# B&R Automation Studio project datmod
Automation Studio 4.3.6.57 SP; Default project

## Configuration Simulation

CPU , AutomationRuntime G4.34, Build 4.1.2, Vc V4.34.2

### Task classes (Cpu.sw)
```
Cyclic#1 (cycle 100000 us, tolerance 10000000 us):
  recipe <- recipe.prg
Binaries: ashwd, sysconf, asfw, arconfig, iomap
Libraries: AsIecCon, astime, datmodHand, DataObj, runtime
```

### Hardware
```
PLC1 : PC_any v1.1.0.0 (OrderNumber=PC)
  VolatileGlobalPvSize = 4096
  XLinkUseDefault = 0
  Cyclic1Duration = 100000
  Cyclic1Tolerance = 10000000
  Cyclic2Duration = 200000
  Cyclic2Tolerance = 10000000
  Cyclic3Duration = 500000
  Cyclic3Tolerance = 10000000
  Cyclic4Duration = 1000000
  Cyclic4Tolerance = 10000000
  Cyclic5Duration = 2000000
  Cyclic5Tolerance = 10000000
  Cyclic6Duration = 3000000
  Cyclic6Tolerance = 12000000
  Cyclic7Duration = 4000000
  Cyclic7Tolerance = 12000000
  Cyclic8Duration = 5000000
  Cyclic8Tolerance = 30000000
```

## Logical view

Binary libraries used (declarations not repeated): DataObj, Runtime, Operator, AsIecCon, astime

### Program Logical/recipe (IEC) - sample program

#### recipe.st - Implementation code
```iecst
PROGRAM _INIT

recipe1.milk := 0.4;
recipe1.name := 'espresso';
recipe1.sugar := 1;

//
END_PROGRAM

PROGRAM _CYCLIC

	CASE step OF
		0: (* store data *)
		recipeHandling.para.pData := ADR(recipe1);
		recipeHandling.para.dataLen := SIZEOF(recipe1);
		recipeHandling.para.memType := doUSRROM;
		recipeHandling.para.name := 'recipe00';
		recipeHandling.para.overwriteExisting := 1;
		recipeHandling.cmd.save := 1;
		step := 1;

		1: (* load data *)
		IF recipeHandling.status.ok THEN
			recipeHandling.para.pData := ADR(recipe2);
			recipeHandling.para.dataLen := SIZEOF(recipe1);
			recipeHandling.para.memType := doUSRROM;
			recipeHandling.para.name := 'recipe00';
			recipeHandling.cmd.load := 1;
			step := 2;
		END_IF

		2:

	END_CASE

	(* call function *)
	datmodHand( recipeHandling );

END_PROGRAM
```

#### recipe.typ - Local data types
```iecst
TYPE
	myRecipe : 	STRUCT
		sugar : USINT;
		milk : REAL;
		name : STRING[20];
	END_STRUCT;
END_TYPE
```

#### recipe.var - Local variables
```iecst
VAR
	step : USINT := 0;
	recipe2 : myRecipe := (0);
	recipe1 : myRecipe := (0);
	recipeHandling : datmodHand_typ := (0);
END_VAR
```

### Package Logical/Libraries - Global libraries

### Library Logical/Libraries/datmodHand (IEC) - simple data module handling

#### datmodHand.typ - Exported data types
```iecst
TYPE
	datmodHandPara_typ : 	STRUCT
		name : STRING[10]; (*name of data module*)
		overwriteExisting : BOOL; (*overwrite existing module*)
		pData : UDINT; (*pointer to data buffer*)
		dataLen : UDINT; (*length of data*)
		memType : USINT; (*target memory in which the data object is to be saved,  e.g. doTEMP, doUSRRAM, doUSRROM, ...*)
	END_STRUCT;
	datmodHandCmd_typ : 	STRUCT  (*1 = execute, 2 = busy*)
		load : BOOL; (*load module*)
		save : BOOL; (*save data to module*)
		delete : BOOL; (*delete module*)
	END_STRUCT;
	datmodHandStatusError_typ : 	STRUCT
		AlreadyExist : BOOL; (*module already exist*)
		NotFound : BOOL; (*module not found*)
		WrongParameter : BOOL; (*parameter error (e.g. para.dataLen = 0, para.pData = 0, para.name = '' )*)
	END_STRUCT;
	datmodHandStatus_typ : 	STRUCT
		ok : BOOL; (*command executed with no error*)
		error : datmodHandStatusError_typ; (*command executed with errors*)
		busy : BOOL; (*busy*)
	END_STRUCT;
	datmodHandInternal_typ : 	STRUCT
		step : UINT;
		fubObjCreate : DatObjCreate;
		fubObjDelete : DatObjDelete;
		fubObjInfo : DatObjInfo;
		fubObjRead : DatObjRead;
	END_STRUCT;
	datmodHand_typ : 	STRUCT
		cmd : datmodHandCmd_typ; (*commands*)
		para : datmodHandPara_typ; (*parameters*)
		status : datmodHandStatus_typ; (*states*)
		internal : datmodHandInternal_typ; (*(internal use)*)
	END_STRUCT;
END_TYPE
```

#### datmodHand.st - data module handling
```iecst
 (* data module handling *)
FUNCTION datmodHand
	datmodHand := 0;
	inst.status.busy := 0;
	CASE inst.internal.step OF
		0: (* wait for command *)
		IF inst.cmd.load = 1 THEN  (* load module *)
			datmodHand := 65535;
			IF inst.para.pData <> 0 AND inst.para.dataLen <> 0  THEN
				inst.status.busy := 1;
				inst.internal.fubObjInfo( enable := 0 );
				inst.status.error.AlreadyExist := 0;
				inst.status.error.NotFound := 0;
				inst.status.error.WrongParameter := 0;
				inst.status.ok := 0;
				inst.internal.step := 10;
			ELSE
				inst.status.error.WrongParameter := 1;
			END_IF
		ELSIF inst.cmd.delete = 1 THEN (* delete module *)
			datmodHand := 65535;
			inst.status.busy := 1;
			inst.internal.fubObjInfo( enable := 0 );
			inst.internal.fubObjDelete( enable := 0 );
			inst.status.error.AlreadyExist := 0;
			inst.status.error.NotFound := 0;
			inst.status.error.WrongParameter := 0;
			inst.status.ok := 0;

			inst.internal.step := 20;
		ELSIF inst.cmd.save = 1 THEN (* save data to module *)
			datmodHand := 65535;
			IF inst.para.pData <> 0 AND inst.para.dataLen <> 0 THEN
				inst.status.busy := 1;
				inst.internal.fubObjCreate( enable := 0 );
				inst.internal.fubObjInfo( enable := 0 );
				inst.internal.fubObjDelete( enable := 0 );
				inst.status.error.AlreadyExist := 0;
				inst.status.error.NotFound := 0;
				inst.status.error.WrongParameter := 0;
				inst.status.ok := 0;
				inst.internal.step := 30;
			ELSE
				inst.status.error.WrongParameter := 1;
			END_IF
		END_IF

		10: (* load *)
		inst.internal.fubObjInfo( enable := 1, pName := ADR(inst.para.name) );
		IF inst.internal.fubObjInfo.status = 0 THEN
			inst.internal.fubObjRead( enable := 1, ident := inst.internal.fubObjInfo.ident, Offset := 0, pDestination := inst.para.pData, len := inst.para.dataLen );
			inst.cmd.load := 0;
			inst.status.ok := 1;
			inst.internal.step := 0;
		ELSIF inst.internal.fubObjInfo.status = doERR_ILLPARAMETER THEN
			inst.cmd.load := 0;
			inst.status.error.WrongParameter := 1;
			inst.internal.step := 0;
		ELSIF inst.internal.fubObjInfo.status = doERR_ILLOBJTYPE OR inst.internal.fubObjInfo.status = doERR_MODULNOTFOUND THEN
			inst.cmd.load := 0;
			inst.status.error.NotFound := 1;
			inst.internal.step := 0;

		END_IF

		20: (* delete *)
		inst.internal.fubObjInfo( enable := 1, pName := ADR(inst.para.name) );
		IF inst.internal.fubObjInfo.status = 0 THEN
			inst.internal.fubObjDelete( enable := 1, ident := inst.internal.fubObjInfo.ident );
			inst.internal.step := 21;
		ELSIF inst.internal.fubObjInfo.status = doERR_ILLPARAMETER THEN
			inst.cmd.delete := 0;
			inst.status.error.WrongParameter := 1;
			inst.internal.step := 0;
		ELSIF inst.internal.fubObjInfo.status = doERR_ILLOBJTYPE OR inst.internal.fubObjInfo.status = doERR_MODULNOTFOUND THEN
			inst.cmd.delete := 0;
			inst.status.error.NotFound := 1;
			inst.internal.step := 0;
		END_IF

		21:
		IF inst.internal.fubObjDelete.status = 0 THEN
			inst.cmd.delete := 0;
			inst.status.ok := 1;
			inst.internal.step := 0;
		ELSIF inst.internal.fubObjDelete.status <> 65535 THEN
			inst.cmd.delete := 0;
			inst.status.error.NotFound := 1;
			inst.internal.step := 0;
		ELSE
			inst.internal.fubObjDelete();
		END_IF

		30: (* save *)
		inst.internal.fubObjInfo( enable := 1, pName := ADR(inst.para.name) );
		IF inst.internal.fubObjInfo.status = 0 THEN
			IF inst.para.overwriteExisting = 0 THEN
				inst.cmd.save := 0;
				inst.status.error.AlreadyExist := 1;
				inst.internal.step := 0;
			ELSE
				inst.internal.fubObjDelete( enable := 1, ident := inst.internal.fubObjInfo.ident );
				inst.internal.step := 31; (* module found ==> delete *)
			END_IF
		ELSIF inst.internal.fubObjInfo.status = doERR_ILLPARAMETER THEN
			inst.cmd.save := 0;
			inst.status.error.WrongParameter := 1;
			inst.internal.step := 0;
		ELSIF inst.internal.fubObjInfo.status = doERR_ILLOBJTYPE OR inst.internal.fubObjInfo.status = doERR_MODULNOTFOUND THEN
			inst.internal.step := 32;  (* module not found ==> create *)
		END_IF

		31:  (* module found ==> delete *)
		IF inst.internal.fubObjDelete.status = 0 THEN
			inst.internal.step := 32;
		ELSIF inst.internal.fubObjDelete.status <> 65535 THEN
			inst.cmd.save := 0;
			inst.status.error.NotFound := 1;
			inst.internal.step := 0;
		ELSE
			inst.internal.fubObjDelete();
		END_IF

		32:  (* create module *)
		inst.internal.fubObjCreate( enable := 1, pName := ADR(inst.para.name), grp := 0, len:= inst.para.dataLen, MemType := inst.para.memType, pCpyData := inst.para.pData );
		IF inst.internal.fubObjCreate.status = 0 THEN
			inst.cmd.save := 0;
			inst.status.ok := 1;
			inst.internal.step := 0;
		ELSIF inst.internal.fubObjCreate.status = doERR_ILLPARAMETER THEN
			inst.cmd.save := 0;
			inst.status.error.WrongParameter := 1;
			inst.internal.step := 0;
		ELSIF inst.internal.fubObjCreate.status <> 65535 THEN
			inst.cmd.save := 0;
			inst.status.error.NotFound := 1;
			inst.internal.step := 0;
		ELSE
			inst.internal.fubObjCreate();
		END_IF

	END_CASE
END_FUNCTION
```

#### datmodHand.fun - Exported functions and function blocks
```iecst
FUNCTION datmodHand : UINT (*data module handling*)
	VAR_INPUT
		inst : datmodHand_typ;
	END_VAR
END_FUNCTION
```
